FUNCTION_BLOCK FB_TransportA
VAR_INPUT
	bstop1 : BOOL;
	bstop2 : BOOL;
	bstop3 : BOOL;
END_VAR
VAR_OUTPUT
	//Hardware Signale
	bstopper1 : BOOL;
	bstopper2 : BOOL;
	bstopper3 : BOOL;
END_VAR
VAR
END_VAR

bstopper1 := bstop1;
bstopper2 := bstop2;
bstopper3 := bstop3;

END_FUNCTION_BLOCK

(* stored: Version 1.1.0.1, ProductVersion 3.1.4024.15
   POU FB_TransportA: Id {e82230df-1a18-4c7e-9a55-8976c76cd3d2}, SpecialFunc None *)
